// TIA Portal V18 export
DATA_BLOCK "DHWAI"   // DB1400
{ S7_Optimized_Access := 'FALSE' }
VERSION : 0.1
// stored: AutoNumber false, DBAccessibleFromOPCUA true, IsOnlyStoredInLoadMemory false, IsWriteProtectedInAS false
   VAR
      AI { S7_SetPoint := 'True'} : "UDT_WSsAI";
   END_VAR
BEGIN
END_DATA_BLOCK
